Omron CX-Programmer project NewProject (CX-Programmer 9.61)

# PLC NewPLC1: CP1L L

## Global symbols (name address type ; comment)
Main FunctionBlock1

## Program NewProgram1 (cyclic task 0)
Local symbols
ctime 0.10 BOOL

### Section Section1

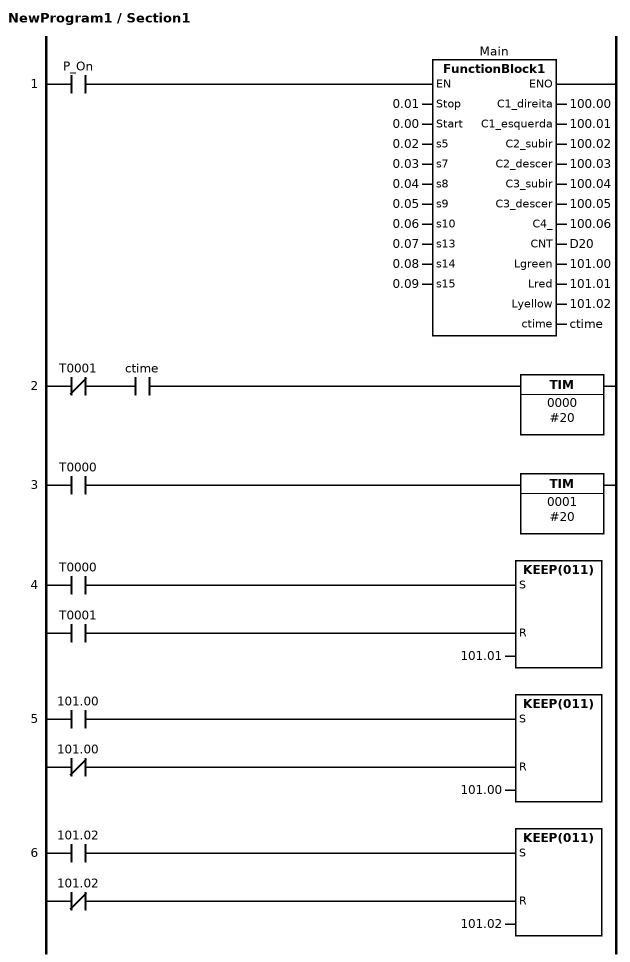
; rung 1
LD P_On
CALL Main : FunctionBlock1 (Stop := 0.01, Start := 0.00, s5 := 0.02, s7 := 0.03, s8 := 0.04, s9 := 0.05, s10 := 0.06, s13 := 0.07, s14 := 0.08, s15 := 0.09, C1_direita => 100.00, C1_esquerda => 100.01, C2_subir => 100.02, C2_descer => 100.03, C3_subir => 100.04, C3_descer => 100.05, C4_ => 100.06, CNT => D20, Lgreen => 101.00, Lred => 101.01, Lyellow => 101.02, ctime => ctime)
; rung 2
LDNOT T0001
AND ctime
TIM 0000 #20
; rung 3
LD T0000
TIM 0001 #20
; rung 4
LD T0000
LD T0001
KEEP(011) 101.01
; rung 5
LD 101.00
LDNOT 101.00
KEEP(011) 101.00
; rung 6
LD 101.02
LDNOT 101.02
KEEP(011) 101.02

### Section END
; rung 0
END(001)

## Function block FunctionBlock1
VAR_INPUT
  Stop : BOOL;
  Start : BOOL;
  s5 : BOOL;
  s7 : BOOL;
  s8 : BOOL := TRUE;
  s9 : BOOL;
  s10 : BOOL := TRUE;
  s13 : BOOL;
  s14 : BOOL;
  s15 : BOOL;
END_VAR
VAR_OUTPUT
  C1_direita : BOOL;
  C1_esquerda : BOOL;
  C2_subir : BOOL;
  C2_descer : BOOL;
  C3_subir : BOOL;
  C3_descer : BOOL;
  C4_ : BOOL;
  CNT : INT;
  Lgreen : BOOL;
  Lred : BOOL;
  Lyellow : BOOL;
  ctime : BOOL;
END_VAR
VAR
  EstadoAtivo : INT;
END_VAR
(*Étapa 0*)
IF ((EstadoAtivo = 0 AND Stop = TRUE) OR (EstadoAtivo = 2 AND s7 = FALSE) OR (EstadoAtivo = 6 AND s7 = FALSE) OR (EstadoAtivo = 11 AND Stop = TRUE) OR
	(EstadoAtivo = 12 AND s5 = FALSE) OR (EstadoAtivo = 13 AND Stop = TRUE) OR ((EstadoAtivo = 14 OR EstadoAtivo = 16 OR EstadoAtivo = 17) AND Stop = TRUE))THEN
	EstadoAtivo := 0;
	C1_direita := FALSE;
	C1_esquerda := FALSE;
	C2_subir := FALSE;
	C2_descer := FALSE;
	C3_subir := FALSE;
	C3_descer := FALSE;
	C4_ := FALSE;
	Lgreen := FALSE;
	Lyellow := FALSE;
	Lred := FALSE;
	ctime:=FALSE;
	CNT := 0;
END_IF;

(*Étapa 1*)
IF((EstadoAtivo = 0 AND Start = TRUE AND Stop = FALSE AND s7 = TRUE AND s15 = TRUE) OR (EstadoAtivo = 14 AND Stop = FALSE AND s15 = TRUE AND s7 = TRUE) OR
	(EstadoAtivo = 15 AND Stop = FALSE AND s15 = TRUE AND s7 = TRUE) OR (EstadoAtivo = 16 AND Start = TRUE AND Stop = FALSE AND s15 = TRUE AND s7 = TRUE))THEN
	EstadoAtivo := 1;
	C1_direita := FALSE;
	C1_esquerda := FALSE;
	C2_subir := FALSE;
	C2_descer := TRUE;
	C3_subir := FALSE;
	C3_descer := FALSE;
	C4_ := FALSE;
	Lred := FALSE;
END_IF;

(*Étapa 2*)
IF((EstadoAtivo = 1 OR EstadoAtivo = 3 OR EstadoAtivo = 9) AND s8 = TRUE AND Stop = TRUE)THEN
	EstadoAtivo := 2;
	C1_direita := FALSE;
	C1_esquerda := FALSE;
	C2_subir := TRUE;
	C2_descer := FALSE;
	C3_subir := FALSE;
	C3_descer := FALSE;
	C4_ := FALSE;
	Lred := FALSE;
END_IF;

(*Étapa 3*)
IF((EstadoAtivo = 1) AND s8 = FALSE AND s5 = TRUE AND Stop = FALSE)THEN
	EstadoAtivo := 3;
	C1_direita := TRUE;
	C1_esquerda := FALSE;
	C2_subir := FALSE;
	C2_descer := FALSE;
	C3_subir := FALSE;
	C3_descer := FALSE;
	C4_ := FALSE;
	Lred := FALSE;
END_IF;

(*Étapa 4*)
IF((EstadoAtivo = 3) AND s13 = TRUE AND s9 = TRUE AND Stop = FALSE)THEN
	EstadoAtivo := 4;
	C1_direita := FALSE;
	C1_esquerda := FALSE;
	C2_subir := FALSE;
	C2_descer := FALSE;
	C3_subir := FALSE;
	C3_descer := TRUE;
	C4_ := FALSE;
	Lred := FALSE;
END_IF;

(*Étapa 5*)
IF((EstadoAtivo = 4 OR EstadoAtivo = 7 OR EstadoAtivo = 8) AND Stop = TRUE AND s10 = TRUE)THEN
	EstadoAtivo := 5;
	C1_direita := FALSE;
	C1_esquerda := FALSE;
	C2_subir := FALSE;
	C2_descer := FALSE;
	C3_subir := TRUE;
	C3_descer := FALSE;
	C4_ := FALSE;
	Lred := FALSE;
END_IF;

(*Étapa 6*)
IF((EstadoAtivo = 5) AND s9 = FALSE AND s8 = TRUE)THEN
	EstadoAtivo := 6;
	C1_direita := FALSE;
	C1_esquerda := FALSE;
	C2_subir := TRUE;
	C2_descer := FALSE;
	C3_subir := FALSE;
	C3_descer := FALSE;
	C4_ := FALSE;
	Lred := FALSE;
END_IF;

(*Étapa 7*)
IF((EstadoAtivo = 4) AND s10 = FALSE AND Stop = FALSE)THEN
	EstadoAtivo := 7;
	C1_direita := FALSE;
	C1_esquerda := FALSE;
	C2_subir := FALSE;
	C2_descer := FALSE;
	C3_subir := FALSE;
	C3_descer := FALSE;
	C4_ := TRUE;
	Lred := FALSE;
END_IF;

(*Étapa 8*)
IF((EstadoAtivo = 7) AND s13 = FALSE AND s14 = TRUE AND Stop = FALSE )THEN
	EstadoAtivo := 8;
	C1_direita := FALSE;
	C1_esquerda := FALSE;
	C2_subir := FALSE;
	C2_descer := FALSE;
	C3_subir := FALSE;
	C3_descer := FALSE;
	C4_ := FALSE;
	CNT := CNT+1;
	Lred := FALSE;
END_IF;

(*Étapa 9*)
IF((EstadoAtivo = 8) AND s10 = TRUE AND s14 = FALSE AND Stop =FALSE)THEN
	EstadoAtivo := 9;
	C1_direita := FALSE;
	C1_esquerda := FALSE;
	C2_subir := FALSE;
	C2_descer := FALSE;
	C3_subir := TRUE;
	C3_descer := FALSE;
	C4_ := FALSE;
	Lred := FALSE;
END_IF;

(*Étapa 10*)
IF((EstadoAtivo = 9) AND s9 = FALSE AND s8 = TRUE AND Stop = FALSE)THEN
	EstadoAtivo := 10;
	C1_direita := FALSE;
	C1_esquerda := FALSE;
	C2_subir := TRUE;
	C2_descer := FALSE;
	C3_subir := FALSE;
	C3_descer := FALSE;
	C4_ := FALSE;
	Lred := FALSE;
END_IF;

(*Étapa 11*)
IF((EstadoAtivo = 10) AND s7 = FALSE AND Stop = FALSE)THEN
	EstadoAtivo := 11;
	C1_direita := FALSE;
	C1_esquerda := TRUE;
	C2_subir := FALSE;
	C2_descer := FALSE;
	C3_subir := FALSE;
	C3_descer := FALSE;
	C4_ := FALSE;
	Lred := FALSE;
END_IF;

(*Étapa 12*)
IF((EstadoAtivo = 10)  AND Stop = TRUE)THEN
	EstadoAtivo := 12;
	C1_direita := FALSE;
	C1_esquerda := TRUE;
	C2_subir := FALSE;
	C2_descer := FALSE;
	C3_subir := FALSE;
	C3_descer := FALSE;
	C4_ := FALSE;
	Lred := FALSE;
END_IF;

(*Étapa 13*)
IF((EstadoAtivo = 11)  AND Stop = FALSE AND s5 = FALSE)THEN
	EstadoAtivo := 13;
	C1_direita := FALSE;
	C1_esquerda := FALSE;
	C2_subir := FALSE;
	C2_descer := FALSE;
	C3_subir := FALSE;
	C3_descer := FALSE;
	C4_ := FALSE;
	Lred := FALSE;
END_IF;

(*Étapa 14*)
IF((EstadoAtivo = 13) AND CNT < 8 AND Stop = FALSE)THEN
	EstadoAtivo := 14;
	C1_direita := FALSE;
	C1_esquerda := FALSE;
	C2_subir := FALSE;
	C2_descer := FALSE;
	C3_subir := FALSE;
	C3_descer := FALSE;
	C4_ := FALSE;
	Lgreen := TRUE;
	Lyellow := FALSE;
	Lred := FALSE;
END_IF;

(*Étapa 15*)
IF((EstadoAtivo = 13) AND CNT >=8  AND CNT <10 AND Stop = FALSE)THEN
	EstadoAtivo := 15;
	C1_direita := FALSE;
	C1_esquerda := FALSE;
	C2_subir := FALSE;
	C2_descer := FALSE;
	C3_subir := FALSE;
	C3_descer := FALSE;
	C4_ := FALSE;
	Lgreen := FALSE;
	Lyellow := TRUE;
	Lred := FALSE;
END_IF;

(*Étapa 16*)
IF((EstadoAtivo = 13) AND CNT = 10 AND Stop = FALSE)THEN
	EstadoAtivo := 16;
	C1_direita := FALSE;
	C1_esquerda := FALSE;
	C2_subir := FALSE;
	C2_descer := FALSE;
	C3_subir := FALSE;
	C3_descer := FALSE;
	C4_ := FALSE;
	Lgreen := FALSE;
	Lyellow := FALSE;
	ctime :=  TRUE;
END_IF;